(* CoDeSys 2.3 export: FC_MQTT_COPYTELEGRAM_V10.EXP *)

(* POU _Generic/Mqtt/Intern/FC_Mqtt_CopyTelegram_V10, ST *)
FUNCTION FC_Mqtt_CopyTelegram_V10 : BOOL
VAR_IN_OUT
	stMqttSrcTelegram	: ST_MqttTelegram;
	stMqttDestTelegram	: ST_MqttTelegram;
	stMqttSettings		: ST_MqttSettings;
END_VAR
VAR
END_VAR
MEMCPY(
	destAddr	:= ADR(stMqttDestTelegram.arMqttData),
    srcAddr		:= ADR(stMqttSrcTelegram.arMqttData),
	n  			:= stMqttSettings.iTelegramSize
);

stMqttDestTelegram.nDataLength := stMqttSrcTelegram.nDataLength;
END_FUNCTION
